FUNCTION_BLOCK TmsHoldStation EXTENDS Process
VAR_INPUT
END_VAR
VAR_OUTPUT
END_VAR
VAR
END_VAR

METHOD PUBLIC MoverArriving : BOOL
VAR_INPUT
	mover : IMover;
END_VAR
VAR
	iTmsMover : ITmsMover;
END_VAR
IF StationMovers <= 2 THEN
	StationMovers := StationMovers + 1;
	IF __QUERYINTERFACE(mover,iTmsMover) THEN
		movers[StationMovers] := iTmsMover;
	END_IF
END_IF
END_METHOD

END_FUNCTION_BLOCK

(* stored: Version 1.1.0.1, ProductVersion 3.1.4024.11
   POU TmsHoldStation: Id {27770a69-a787-45d0-98d5-3048dc805328}, SpecialFunc None
   Method MoverArriving: Id {9da69018-e0b3-43b6-8b40-80f26b1bd5d9} *)
